{attribute 'to_string'}
TYPE E_RmtInCtrl :
(
	None := 0,
	Remote1,
	Remote2
);
END_TYPE

(* stored: Version 1.1.0.1, ProductVersion 3.1.4026.18
   DUT E_RmtInCtrl: Id {2e65cad9-45c1-47f9-a9fb-e508ba895143} *)
